// Mitsubishi GX Works2 project: teste 28   PLC: Q03UDV

PROGRAM MAIN
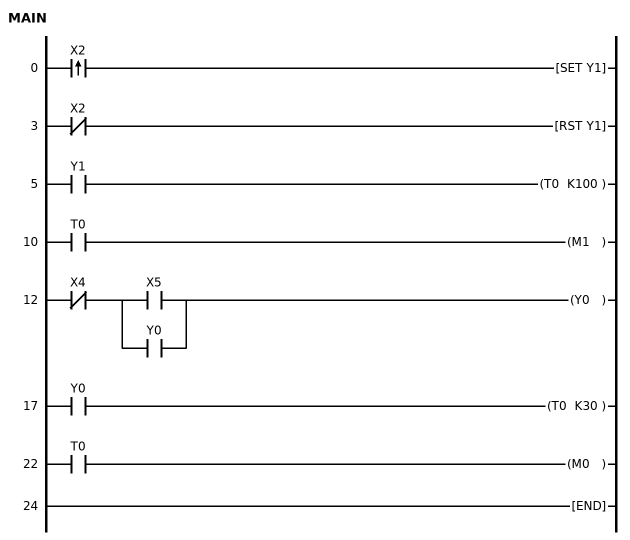
0     LDP     X2
      SET     Y1
3     LDI     X2
      RST     Y1
5     LD      Y1
      OUT     T0 K100
10    LD      T0
      OUT     M1
12    LDI     X4
      LD      X5
      OR      Y0
      ANB
      OUT     Y0
17    LD      Y0
      OUT     T0 K30
22    LD      T0
      OUT     M0
24    END
END_PROGRAM
